TYPE U_UMC_Lenze_Control :

UNION
	Output: UINT;
	Data: T_UMC_Lenze_Control;
END_UNION

END_TYPE

(* stored: Version 1.1.0.1, ProductVersion 3.1.0.26
   DUT U_UMC_Lenze_Control: Id {9768d289-6cef-41e2-82ba-11dc57e84170} *)
